Staubli VAL3: getJointDate.pgx

program getJointDate(string x_sText (dimensions=1), jointRx& x_jJoint (dimensions=1))
  local string l_sJntDate[6]
  local bool l_bBool
begin
  call split(x_sText,",",l_sJntDate)
  l_sJntDate[0]=toNum(l_sJntDate[0],x_jJoint.j1,l_bBool)
  l_sJntDate[1]=toNum(l_sJntDate[1],x_jJoint.j2,l_bBool)
  l_sJntDate[2]=toNum(l_sJntDate[2],x_jJoint.j3,l_bBool)
  l_sJntDate[3]=toNum(l_sJntDate[3],x_jJoint.j4,l_bBool)
  l_sJntDate[4]=toNum(l_sJntDate[4],x_jJoint.j5,l_bBool)
  l_sJntDate[5]=toNum(l_sJntDate[5],x_jJoint.j6,l_bBool)

end
